Staubli VAL3: init.pgx

public program init()
begin
  //主轴工具:停止
  dioSet(doB_7_toolOn,0)
  //转台:停止
  dioSet(doB_9_tableOn,0)

end
